FUNCTION_BLOCK GroupShutterSwitch
VAR_INPUT
END_VAR
VAR_OUTPUT
END_VAR
VAR
END_VAR

END_FUNCTION_BLOCK

(* stored: Version 1.1.0.1, ProductVersion 3.1.4024.12
   POU GroupShutterSwitch: Id {9aebf698-8609-4143-8f8a-6a4a1a3cf539}, SpecialFunc None *)
